RoboDK station: Stringer A-BotUP-BOX1.rdk

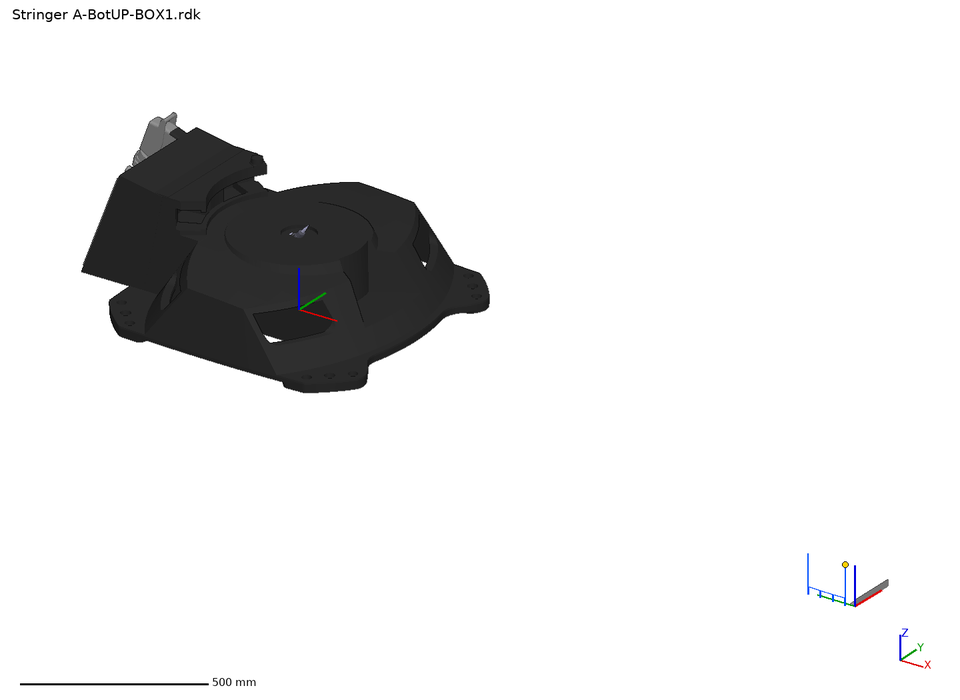
[picture v0: the station drawn from its stored meshes, robots at their saved joint values, targets as dots, program paths as lines]
Station Stringer A-BotUP-BOX1 (saved by RoboDK 5.2.3). Poses are relative to the parent item; angles as X-Y-Z fixed-axis rotations.
  - frame KUKA KR 210 R2700 extra Base at (0, 0, 0) mm
    - robot KUKA KR 210 R2700 extra: 6 axes, payload 210 kg, reach 2696 mm, repeatability 0.06 mm, weight 1068 kg
        joint limits [-185, -140, -120, -350, -125, -350] to [185, -5, 155, 350, 125, 350]; home [0, -90, 90, 0, 0, 0]; saved at [-5.485, -33.945, 111.477, 172.283, 26.612, -177.36]
      - tool Spindle, TCP at (32, 0, 260) mm, rotated rx 0 ry 39 rz 0 deg, size 157.3 x 72 x 259.9 mm
  - frame Frame 2 at (1800, 0, -372.68) mm, rotated rx 0 ry 0 rz 90 deg
    - object Stringer A-BotUP-BOX1 at (0, 0, 0) mm, rotated rx 0 ry 0 rz -90 deg, 4 curves, geometry from Point 4
    - object L-Stringer A - bot up at (0, 0, 0) mm, size 162.3 x 20 x 20 mm, geometry from L-Stringer A - bot up.stl
  - machining project Point settings: rotZ(0) | rotX(0)*rotY(0) | rotz(0) | onStart | onPathStart | onApproach | onPoint | onRetract | onFinish | SetRPM(%1) | SetTool(%1) | Extruder(%1) | default | default | OutOnMov(%1) | OutOffMov(%1) | onPathFinish | M_RunCode(%1)
  - program Point (31 instructions, listed below)
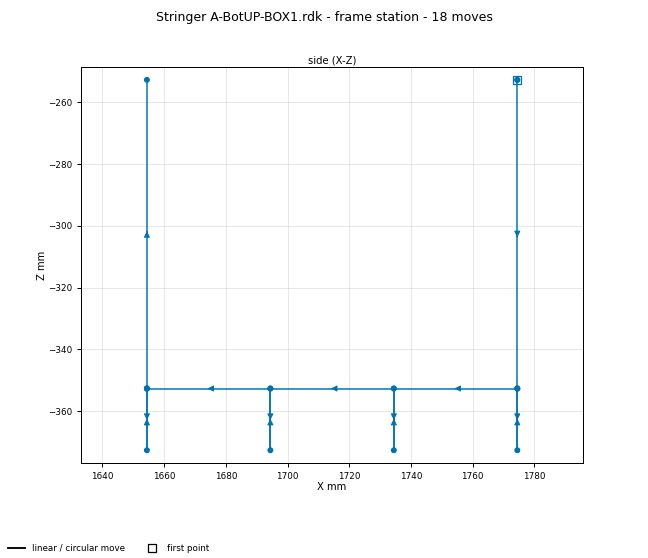
[picture p0: tool path of Stringer A-BotUP-BOX1.rdk in frame station, 18 of 18 moves have a stored position in this frame; points joined in program order, loops and branches not executed]

--- program Point (robot KUKA KR 210 R2700 extra) ---
  Smooth(1)
  Set speed (1000.0 mm/s)
  Set Ref.: Frame 2
  Set Tool: Spindle
  Show Spindle
  MoveJ 1 to (-9.87, 25.57, 120) mm, rotated rx -180 ry 0 rz -180 deg; joints [-0.966, -34.011, 111.835, 178.653, 26.827, -179.548]
  MoveL 2 to (-9.87, 25.57, 120) mm, rotated rx -180 ry 0 rz -180 deg; joints [-0.966, -34.011, 111.835, 178.653, 26.827, -179.548]
  MoveL 3 to (-9.87, 25.57, 20) mm, rotated rx -180 ry 0 rz -180 deg; joints [-0.966, -28.682, 109.193, 178.766, 29.512, -179.677]
  MoveL 4 to (-9.87, 25.57, 20) mm, rotated rx -180 ry 0 rz -180 deg; joints [-0.966, -28.682, 109.193, 178.766, 29.512, -179.677]
  Set speed (50.0 mm/s)
  MoveL 5 to (-9.87, 25.57, 0) mm, rotated rx 180 ry 0 rz 180 deg; joints [-0.966, -27.624, 108.617, 178.784, 29.994, -179.697]
  MoveL 6 to (-9.87, 25.57, 20) mm, rotated rx -180 ry 0 rz -180 deg; joints [-0.966, -28.682, 109.193, 178.766, 29.512, -179.677]
  Set speed (1000.0 mm/s)
  MoveL 7 to (-9.87, 65.57, 20) mm, rotated rx 180 ry 0 rz 180 deg; joints [-2.476, -28.674, 109.13, 176.831, 29.468, -179.166]
  Set speed (50.0 mm/s)
  MoveL 8 to (-9.87, 65.57, 0) mm, rotated rx 180 ry 0 rz 180 deg; joints [-2.476, -27.616, 108.555, 176.878, 29.949, -179.219]
  MoveL 9 to (-9.87, 65.57, 20) mm, rotated rx 180 ry 0 rz 180 deg; joints [-2.476, -28.674, 109.13, 176.831, 29.468, -179.166]
  Set speed (1000.0 mm/s)
  MoveL 10 to (-9.87, 105.57, 20) mm, rotated rx 180 ry 0 rz 180 deg; joints [-3.983, -28.658, 109.013, 174.889, 29.385, -178.641]
  Set speed (50.0 mm/s)
  MoveL 11 to (-9.87, 105.57, 0) mm, rotated rx 180 ry 0 rz -180 deg; joints [-3.983, -27.601, 108.438, 174.963, 29.865, -178.727]
  MoveL 12 to (-9.87, 105.57, 20) mm, rotated rx 180 ry 0 rz 180 deg; joints [-3.983, -28.658, 109.013, 174.889, 29.385, -178.641]
  Set speed (1000.0 mm/s)
  MoveL 13 to (-9.87, 145.57, 20) mm, rotated rx -180 ry 0 rz -180 deg; joints [-5.485, -28.634, 108.842, 172.932, 29.265, -178.094]
  Set speed (50.0 mm/s)
  MoveL 14 to (-9.87, 145.57, 0) mm, rotated rx -180 ry 0 rz -180 deg; joints [-5.485, -27.579, 108.267, 173.036, 29.742, -178.213]
  MoveL 15 to (-9.87, 145.57, 20) mm, rotated rx -180 ry 0 rz -180 deg; joints [-5.485, -28.634, 108.842, 172.932, 29.265, -178.094]
  MoveL 16 to (-9.87, 145.57, 20) mm, rotated rx -180 ry 0 rz -180 deg; joints [-5.485, -28.634, 108.842, 172.932, 29.265, -178.094]
  Set speed (1000.0 mm/s)
  MoveL 17 to (-9.87, 145.57, 20) mm, rotated rx -180 ry 0 rz -180 deg; joints [-5.485, -28.634, 108.842, 172.932, 29.265, -178.094]
  MoveL 18 to (-9.87, 145.57, 120) mm, rotated rx -180 ry 0 rz -180 deg; joints [-5.485, -33.945, 111.477, 172.283, 26.612, -177.36]
